// TIA Portal project "OR" (V17)

(* hardware
DEVICE "S7-1200 station_1"  S7-1200 Station
   slot 0: "Rack_0"  S7-1200 Rack  Rack  V1.0
   slot 1: "PLC_1"  CPU 1212C AC/DC/Rly  6ES7 212-1BE40-0XB0  V4.4
*)

// ===== PLC "PLC_1"  CPU 1212C AC/DC/Rly =====

VAR_GLOBAL   // PLC tag table "Default tag table"
   "Tag_1" AT %I0.0 : Bool;
   "Tag_2" AT %Q0.0 : Bool;
   "System_Byte" AT %MB20 : Byte;
   "FirstScan" AT %M20.0 : Bool;
   "DiagStatusUpdate" AT %M20.1 : Bool;
   "AlwaysTRUE" AT %M20.2 : Bool;
   "AlwaysFALSE" AT %M20.3 : Bool;
   "Clock_Byte" AT %MB25 : Byte;
   "Clock_10Hz" AT %M25.0 : Bool;
   "Clock_5Hz" AT %M25.1 : Bool;
   "Clock_2.5Hz" AT %M25.2 : Bool;
   "Clock_2Hz" AT %M25.3 : Bool;
   "Clock_1.25Hz" AT %M25.4 : Bool;
   "Clock_1Hz" AT %M25.5 : Bool;
   "Clock_0.625Hz" AT %M25.6 : Bool;
   "Clock_0.5Hz" AT %M25.7 : Bool;
   "Tag_3" AT %I0.1 : Bool;
   "Tag_4" AT %QB0 : Byte;
   "Tag_5" AT %I0.2 : Bool;
   "Tag_6" AT %MB2 : Byte;
   "Tag_7" AT %M100.0 : Bool;
   "Tag_8" AT %MW0 : Int;
   "Tag_9" AT %Q0.1 : Bool;
   "Tag_10" AT %Q0.2 : Bool;
   "Tag_11" AT %IW64 : Word;
   "Tag_12" AT %MW10 : Word;
   "Tag_13" AT %MD10 : Real;
END_VAR

ORGANIZATION_BLOCK "Main"   // OB1, LAD, ProgramCycle
TITLE = "Main Program Sweep (Cycle)"
{ S7_Optimized_Access := 'TRUE' }
VERSION : 0.1
   VAR_INPUT
      Initial_Call : Bool;   // Initial call of this OB
      Remanence : Bool;   // =True, if remanent data are available
   END_VAR
BEGIN

REGION Network 1
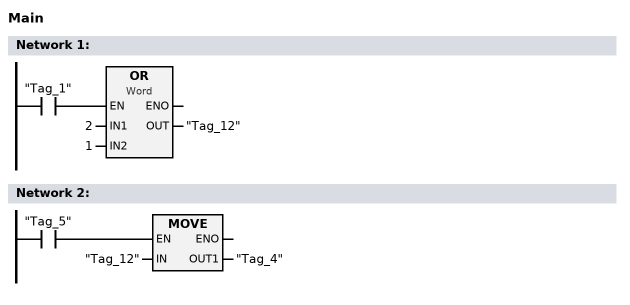
   IF "Tag_1" THEN "Tag_12" := 2 OR 1; END_IF;
END_REGION

REGION Network 2
   RUNG wire#powerrail
      Contact( "Tag_5" )
      Move(in := "Tag_12", out1 => "Tag_4")
   END_RUNG
   // the same network as SCL:
   IF "Tag_5" THEN "Tag_4" := "Tag_12"; END_IF;
END_REGION
END_ORGANIZATION_BLOCK